INTERFACE ITF_GroupE_TE1_HMI_Init EXTENDS ITF_BaseGroupElement, ITF_GroupE_TE1_HMI_Connector

END_INTERFACE

(* stored: Version 1.1.0.1, ProductVersion 3.1.4024.15
   Itf ITF_GroupE_TE1_HMI_Init: Id {0cdc417a-7fd0-4ee9-97e7-633e62c214ae} *)
